FUNCTION_BLOCK FB_SR (* Realizes a bistable set-dominat latch *)
  (* Standard: 61499-1; Description: Copyright (c) 2023 Martin Erich Jobst This program and the accompanying materials are made available under the terms of the Eclipse Public License 2.0 which is available at https://www.eclipse.org/legal/epl-2.0/ SPDX-License-Identifier: EPL-2.0 *)
  (* Version 3.0, 2025-04-14, Patrick Aigner, changed package *)
  (* Version 1.0, 2023-04-28, Martin Jobst *)
  PACKAGE iec61131::bistableElements;
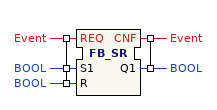
  EVENT_INPUT
    REQ WITH S1, R; (* Normal Execution Request *)
  END_EVENT
  EVENT_OUTPUT
    CNF WITH Q1; (* Execution Confirmation *)
  END_EVENT
  VAR_INPUT
    S1 : BOOL; (* Set *)
    R : BOOL; (* Reset *)
  END_VAR
  VAR_OUTPUT
    Q1 : BOOL; (* Output *)
  END_VAR
  EC_STATES
    REQ : REQ -> CNF;
  END_STATES
  ALGORITHM REQ IN ST:
Q1 := S1 OR ((NOT R) AND Q1);
  END_ALGORITHM
END_FUNCTION_BLOCK
